{attribute 'GeneratedUsingTerminal: ELX3351-0000-0016'}
{attribute addProperty BoxType "ELX3351-0000-0016"}
{attribute addProperty Id "OverrangeBOOL1Data_invalidBOOL1ErrorBOOL1Calibration_in_progressBOOL1Steady_stateBOOL1TxPDO_ToggleBOOL1"}
{attribute addProperty CRC "3514323520"}
{attribute addProperty Size "6"}
TYPE Status_D1785240 :
STRUCT
	{attribute addProperty Name "Overrange"}
	Overrange : BOOL;
	{attribute addProperty Name "Data_invalid"}
	Data_invalid : BOOL;
	{attribute addProperty Name "Error"}
	Error : BOOL;
	{attribute addProperty Name "Calibration_in_progress"}
	Calibration_in_progress : BOOL;
	{attribute addProperty Name "Steady_state"}
	Steady_state : BOOL;
	{attribute addProperty Name "TxPDO_Toggle"}
	TxPDO_Toggle : BOOL;
END_STRUCT
END_TYPE

(* stored: Version 1.2.0.0, ProductVersion 3.1.4024.9
   DUT Status_D1785240: Id {00647a82-8d73-4333-bec1-390d21d24741} *)
